{attribute 'GeneratedUsingTerminal: EL6201-0000-0017'}
{attribute addProperty BoxType "EL6201-0000-0017"}
{attribute addProperty Id "Slave_27A_DI0BOOL1Slave_27A_DI1BOOL1Slave_27A_DI2BOOL1Slave_27A_DI3BOOL1Slave_27B_DI0BOOL1Slave_27B_DI1BOOL1Slave_27B_DI2BOOL1Slave_27B_DI3BOOL1"}
{attribute addProperty CRC "2763941986"}
{attribute addProperty Size "8"}
TYPE Slave_27_Inputs_A4BE6862 :
STRUCT
	{attribute addProperty Name "Slave_27A_DI0"}
	Slave_27A_DI0 : BOOL;
	{attribute addProperty Name "Slave_27A_DI1"}
	Slave_27A_DI1 : BOOL;
	{attribute addProperty Name "Slave_27A_DI2"}
	Slave_27A_DI2 : BOOL;
	{attribute addProperty Name "Slave_27A_DI3"}
	Slave_27A_DI3 : BOOL;
	{attribute addProperty Name "Slave_27B_DI0"}
	Slave_27B_DI0 : BOOL;
	{attribute addProperty Name "Slave_27B_DI1"}
	Slave_27B_DI1 : BOOL;
	{attribute addProperty Name "Slave_27B_DI2"}
	Slave_27B_DI2 : BOOL;
	{attribute addProperty Name "Slave_27B_DI3"}
	Slave_27B_DI3 : BOOL;
END_STRUCT
END_TYPE

(* stored: Version 1.2.0.0, ProductVersion 3.1.4024.9
   DUT Slave_27_Inputs_A4BE6862: Id {473fd9b1-c5ed-47d5-bacb-30b11387bbe0} *)
